(* IEC 61131-3 sources: plc_generation_empirical_study/our_method_delta_DVP48ES300R/calibration/fresh_instance_reset, 1 file *)

(* ---- candidate.st ---- *)
FUNCTION_BLOCK DVP_FRESH_INSTANCE_RESET
VAR_INPUT
    SetLatch : BOOL;
END_VAR
VAR_OUTPUT
    Latched : BOOL;
END_VAR

IF SetLatch THEN
    Latched := TRUE;
END_IF;

END_FUNCTION_BLOCK
